// TIA Portal V20 export
DATA_BLOCK "QDAS_ReadVGageProData"   // DB10000
{ S7_Optimized_Access := 'FALSE' }
// stored: AutoNumber false, InstanceOfName typeReadVGageProData, InstanceOfType UDT
"typeReadVGageProData"
   // VAR
   //    heartbeatActive : Bool;
   //    dataCollected : Bool;
   //    plcOK : Bool;
   //    spareIn_1 : Bool;
   //    spareIn_2 : Bool;
   //    spareIn_3 : Bool;
   //    spareIn_4 : Bool;
   //    spareIn_5 : Bool;
   // END_VAR
BEGIN
END_DATA_BLOCK
